// TwinCAT 3 PLC project MAS418_PLC
// ProgramVersion: 3.1.4024.0
// libraries:
//   Tc2_Standard, * (Beckhoff Automation GmbH)
//   Tc2_System, * (Beckhoff Automation GmbH)
//   Tc3_Module, * (Beckhoff Automation GmbH)
//   VisuDialogs, * (System)
// project tree:
//   / GlobalTextList.TcGTLO, PlcTask.TcTTO, Visualization Manager.TcVMO (not stored)
//   POUs/ MAIN.TcPOU
//   VISUs/ HMI.TcVIS
// real-time tasks:
//   TASK PlcTask: cycle T#10ms, priority 20, ADS port 350

CONFIGURATION MAS418_PLC
    RESOURCE PLC ON TwinCAT3
        TASK PlcTask(INTERVAL := T#10ms, PRIORITY := 20);
        PROGRAM MAIN WITH PlcTask : MAIN;
    END_RESOURCE
END_CONFIGURATION

// ---- POUs/MAIN.TcPOU
PROGRAM MAIN
VAR
	bEnable: BOOL;
	bStart: BOOL;
	nInt: INT:=-32768;
	nUINT:UINT:=65535;
	fREAL: REAL:=255.255;
	sPowerStatus: STRING:='Power off';
	nFloatConversion: INT:= 54;
	fFloatConversion: LREAL;
	nIntConversion: INT;
	fIntConversion: LREAL;
END_VAR

bEnable:=bStart;
fFloatConversion:=nFloatConversion;
//fFloatConversion:= INT_TO_LREAL(nFloatConversion);
nIntConversion:= LREAL_TO_INT(fIntConversion);

END_PROGRAM

// ---- GlobalTextList.TcGTLO
TEXTLIST GlobalTextList
  660 = 'BOOL'
  926 = 'BOOL%i'
  349 = 'DataTypeTesting'
  971 = 'INT'
  568 = 'INT%i'
  137 = 'Power on'
  755 = 'REAL'
  908 = 'REAL%f'
  701 = 'REAL%i'
  350 = 'String'
  365 = 'String%i'
  481 = 'String%s'
  967 = 'UINT'
  72 = 'UINT%i'
END_TEXTLIST

// ---- VISUs/HMI.TcVIS
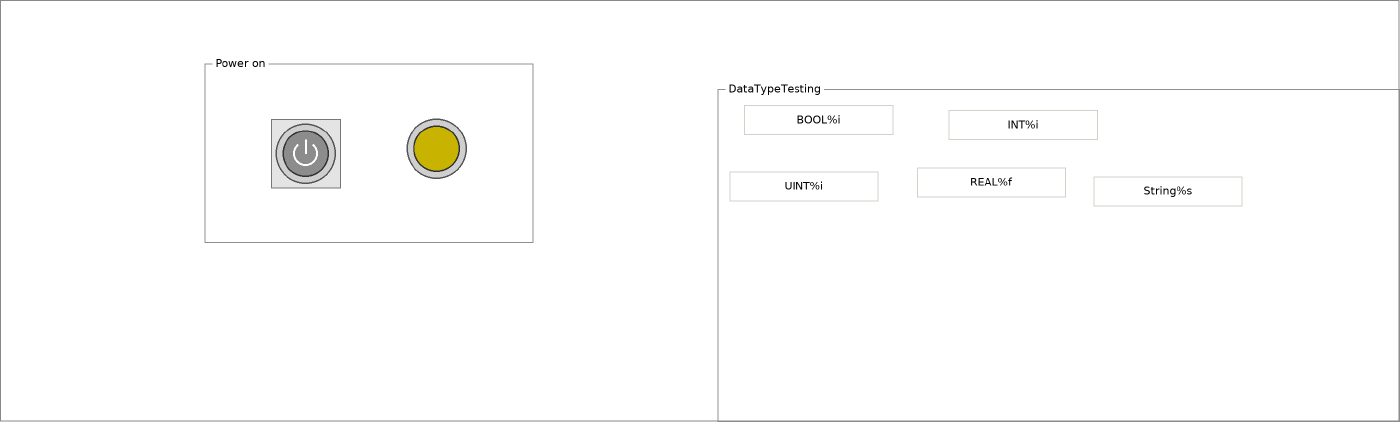
VISUALIZATION HMI  // 1411x426
    GroupBox (206,56 331x189), "Power on"
        PowerSwitch (67,64 70x70), variable: MAIN.bStart, behaviour: TOGGLE, style: Switch-PowerSwitch-Gray
        Lamp1 (199,59 70x70), variable: MAIN.bEnable, style: Lamp-Lamp1-Yellow
    GroupBox (723,82 688x344), "DataTypeTesting"
        Textfield (27,24 150x30), "BOOL%i", text variable: MAIN.bEnable
        Textfield (233,29 150x30), "INT%i", text variable: MAIN.nInt
        Textfield (12,91 150x30), "UINT%i", text variable: MAIN.nUINT
        Textfield (201,87 150x30), "REAL%f", text variable: MAIN.fREAL
            OnMouseDown: write the text variable via Default
        Textfield (379,96 150x30), "String%s", text variable: MAIN.sPowerStatus
            OnMouseDown: write the text variable via Default
END_VISUALIZATION
